TYPE TRunCmdLift :
	(
		RCL_None,
		RCL_MoveToPlate,
		RCL_MoveToLoadPlate,
		RCL_MoveToOpenDrawer
	);
END_TYPE

(* stored: Version 1.1.0.1, ProductVersion 3.1.4022.12
   DUT TRunCmdLift: Id {0fcf46a1-3aec-42dc-83f6-3d66c4f0c30b} *)
